Fanuc KAREL source: kt00928.KL

-- PROVISIONAL review KL for V940-1; original PC SHA256 9283621aafb66992d84e1e2afb5115e51efd0265c09c438837bf184344c1576b
-- Incomplete behavior may be omitted. Consult companion uncertainty JSON. Do not deploy.
PROGRAM KT00928
%NOLOCKGROUP
VAR
  S1 : STRING[80]
  S2 : STRING[80]
  OUT : INTEGER
BEGIN
  -- V9_ZERO_TABLE_METADATA_HINT layout=0001; no indexed target words; source/name/runtime held
  -- UNRESOLVED_PC offsets 5-14; opcodes 3F,75
  -- UNRESOLVED_PC offsets 19-28; opcodes 3F,75
  -- UNRESOLVED_PC offsets 33-42; opcodes 3F,75
  -- UNRESOLVED_PC offsets 47-56; opcodes 3F,75
  -- UNRESOLVED_PC offsets 61-80; opcodes 27,22,2A,27,9D,76,23
  -- UNRESOLVED_PC offsets 85-89; opcodes 7F
END KT00928
